Universal Robots PolyScope program: Tarea_comandos_Adrian.urp

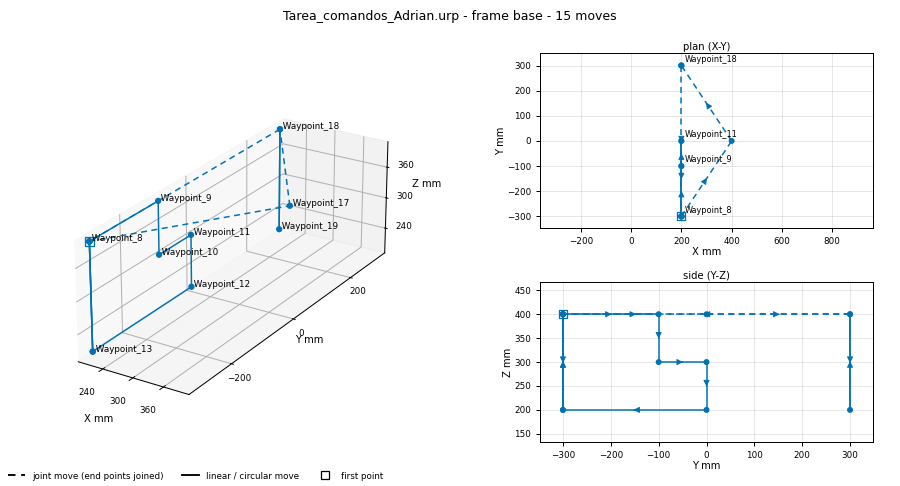
[picture p0: tool path of Tarea_comandos_Adrian.urp in frame base, 15 of 22 moves have a stored position in this frame; points joined in program order, loops and branches not executed]
Program Tarea_comandos_Adrian (installation=default directory=/home/hugo/Documents/Proyecto_Ingenieria/ursim-5.10.2.106319/programs/ASM/Clase1_Comandos createdIn=5.9.4.1031232 lastSavedIn=5.10.2.106319 robotSerialNumber=20195599999)
Calibrated DH parameters: a=[0, -0.425, -0.3922, 0, 0, 0]; d=[0.1625, 0, 0, 0.1333, 0.0997, 0.0996]; alpha=[1.570796, 0, 0, 1.570796, -1.570796, 0]; deltaTheta=[0, 0, 0, 0, 0, 0]
Robot Program (runOnlyOnce=true)
  tipo_trayec :=  (valueSource=Operator message=Tipo de Trayectoria [1,2,3] valueType=Integer)
  num_oper :=  (valueSource=Operator message=Numero de Operaciones valueType=Integer)
  cont_oper := 0
  Loop While (checkContinuously=false) expression=cont_oper<num_oper
    Switch expression=tipo_trayec
      Case (caseValue=1)
        Folder Movimiento1
          MoveL speed 250 mm/s, acceleration 1200 mm/s^2 (useActiveTCP=true) feature=Base
            Waypoint Waypoint_1 (Relative): relativeFromPosition TCP in base x=200 y=-300 z=400 mm, rx=-3.1046 ry=-0.0005 rz=-0.1025 rad; joints [100.772, -111.151, -240.446, -97.122, 274.091, 190.709] deg; TCP in base x=200 y=-300 z=400 mm, rx=-3.1046 ry=-0.0005 rz=-0.1025 rad; joints [100.772, -111.151, -240.446, -97.122, 274.091, 190.709] deg
            Waypoint Waypoint_2 (Relative): relativeFromPosition TCP in base x=200 y=-300 z=400 mm, rx=-3.1046 ry=-0.0005 rz=-0.1025 rad; joints [100.772, -111.151, -240.446, -97.122, 274.091, 190.709] deg; TCP in base x=200 y=-100 z=400 mm, rx=-3.1046 ry=-0.0005 rz=-0.1025 rad; joints [114.432, -137.69, -229.814, -82.219, 274.278, 204.404] deg
            Waypoint Waypoint_3 (Relative): relativeFromPosition TCP in base x=200 y=-100 z=400 mm, rx=-3.1046 ry=-0.0005 rz=-0.1025 rad; joints [114.432, -137.69, -229.814, -82.219, 274.278, 204.404] deg; TCP in base x=200 y=-100 z=300 mm, rx=-3.1046 ry=-0.0005 rz=-0.1025 rad; joints [114.432, -137.762, -215.151, -96.809, 274.278, 204.404] deg
            Waypoint Waypoint_4 (Relative): relativeFromPosition TCP in base x=200 y=-100 z=300 mm, rx=-3.1046 ry=-0.0005 rz=-0.1025 rad; joints [114.432, -137.762, -215.151, -96.809, 274.278, 204.404] deg; TCP in base x=200 y=0 z=300 mm, rx=-3.1046 ry=-0.0005 rz=-0.1025 rad; joints [135.409, -145.831, -213.571, -91.873, 274.093, 225.437] deg
            Waypoint Waypoint_5 (Relative): relativeFromPosition TCP in base x=200 y=0 z=300 mm, rx=-3.1046 ry=-0.0005 rz=-0.1025 rad; joints [135.409, -145.831, -213.571, -91.873, 274.093, 225.437] deg; TCP in base x=200 y=0 z=200 mm, rx=-3.1046 ry=-0.0005 rz=-0.1025 rad; joints [135.409, -140.302, -199.274, -111.698, 274.093, 225.437] deg
            Waypoint Waypoint_6 (Relative): relativeFromPosition TCP in base x=200 y=0 z=200 mm, rx=-3.1046 ry=-0.0005 rz=-0.1025 rad; joints [135.409, -140.302, -199.274, -111.698, 274.093, 225.437] deg; TCP in base x=200 y=-300 z=200 mm, rx=-3.1046 ry=-0.0005 rz=-0.1025 rad; joints [100.772, -94.771, -218.732, -135.215, 274.091, 190.709] deg
            Waypoint Waypoint_7 (Relative): relativeFromPosition TCP in base x=200 y=-300 z=200 mm, rx=-3.1046 ry=-0.0005 rz=-0.1025 rad; joints [100.772, -94.771, -218.732, -135.215, 274.091, 190.709] deg; TCP in base x=200 y=-300 z=400 mm, rx=-3.1046 ry=-0.0005 rz=-0.1025 rad; joints [100.772, -111.151, -240.446, -97.122, 274.091, 190.709] deg
      Case (caseValue=2)
        Folder Movimiento2
          MoveL speed 250 mm/s, acceleration 1200 mm/s^2 (useActiveTCP=true) feature=Base
            Waypoint Waypoint_8: TCP in base x=200 y=-300 z=400 mm, rx=-3.1046 ry=-0.0005 rz=-0.1025 rad; joints [100.772, -111.151, -240.446, -97.122, 274.091, 190.709] deg
            Waypoint Waypoint_9: motionParameters(blendRadius=0.05); TCP in base x=200 y=-100 z=400 mm, rx=-3.1046 ry=-0.0005 rz=-0.1025 rad; joints [114.432, -137.69, -229.814, -82.219, 274.278, 204.404] deg
            Waypoint Waypoint_10: motionParameters(blendRadius=0.05); TCP in base x=200 y=-100 z=300 mm, rx=-3.1046 ry=-0.0005 rz=-0.1025 rad; joints [114.432, -137.762, -215.151, -96.809, 274.278, 204.404] deg
            Waypoint Waypoint_11: motionParameters(blendRadius=0.05); TCP in base x=200 y=0 z=300 mm, rx=-3.1046 ry=-0.0005 rz=-0.1025 rad; joints [135.409, -145.831, -213.571, -91.873, 274.093, 225.437] deg
            Waypoint Waypoint_12: TCP in base x=200 y=0 z=200 mm, rx=-3.1046 ry=-0.0005 rz=-0.1025 rad; joints [135.409, -140.302, -199.274, -111.698, 274.093, 225.437] deg
            Waypoint Waypoint_13: motionParameters(blendRadius=0.05); TCP in base x=200 y=-300 z=200 mm, rx=-3.1046 ry=-0.0005 rz=-0.1025 rad; joints [100.772, -94.771, -218.732, -135.215, 274.091, 190.709] deg
            Waypoint Waypoint_14: TCP in base x=200 y=-300 z=400 mm, rx=-3.1046 ry=-0.0005 rz=-0.1025 rad; joints [100.772, -111.151, -240.446, -97.122, 274.091, 190.709] deg
      Case (caseValue=3)
        Folder Movimiento3
          MoveL speed 250 mm/s, acceleration 1200 mm/s^2 (useActiveTCP=true) feature=Base
            Waypoint Waypoint_15: TCP in base x=200 y=-300 z=400 mm, rx=-3.1046 ry=-0.0005 rz=-0.1025 rad; joints [100.772, -111.151, -240.446, -97.122, 274.091, 190.709] deg; TCP offset x=0 y=0 z=0 mm, rx=0 ry=0 rz=0 rad
            Waypoint Waypoint_16: TCP in base x=200 y=-300 z=200 mm, rx=-3.1046 ry=-0.0005 rz=-0.1025 rad; joints [100.772, -94.771, -218.732, -135.215, 274.091, 190.709] deg
            Waypoint Waypoint_15: TCP in base x=200 y=-300 z=400 mm, rx=-3.1046 ry=-0.0005 rz=-0.1025 rad; joints [100.772, -111.151, -240.446, -97.122, 274.091, 190.709] deg; TCP offset x=0 y=0 z=0 mm, rx=0 ry=0 rz=0 rad
          MoveJ speed 60 deg/s, acceleration 80 deg/s^2 (useActiveTCP=true) feature=Base
            Waypoint Waypoint_17: TCP in base x=400 y=0 z=400 mm, rx=-3.1046 ry=-0.0005 rz=-0.1025 rad; joints [159.685, -105.537, -243.051, -104.258, 273.207, 249.747] deg
          Popup Message (haltProgram=false message=¿Salir de la estacion? inputType=Text)
          MoveJ speed 60 deg/s, acceleration 80 deg/s^2 (useActiveTCP=true) feature=Base
            Waypoint Waypoint_18: TCP in base x=200 y=300 z=400 mm, rx=-3.1046 ry=-0.0005 rz=-0.1025 rad; joints [214.759, -111.86, -238.597, -103.801, 269.506, 304.723] deg
          MoveL speed 250 mm/s, acceleration 1200 mm/s^2 (useActiveTCP=true) feature=Base
            Waypoint Waypoint_19: TCP in base x=200 y=300 z=200 mm, rx=-3.1046 ry=-0.0005 rz=-0.1025 rad; joints [214.759, -94.116, -217.219, -142.923, 269.506, 304.723] deg
            Waypoint Waypoint_18: TCP in base x=200 y=300 z=400 mm, rx=-3.1046 ry=-0.0005 rz=-0.1025 rad; joints [214.759, -111.86, -238.597, -103.801, 269.506, 304.723] deg
          MoveJ speed 60 deg/s, acceleration 80 deg/s^2 (useActiveTCP=true) feature=Base
            Waypoint Waypoint_15: TCP in base x=200 y=-300 z=400 mm, rx=-3.1046 ry=-0.0005 rz=-0.1025 rad; joints [100.772, -111.151, -240.446, -97.122, 274.091, 190.709] deg; TCP offset x=0 y=0 z=0 mm, rx=0 ry=0 rz=0 rad
    cont_oper := cont_oper+1
